// TwinCAT 3 PLC project PLC1
// ProgramVersion: 3.1.4026.16
// libraries:
//   Tc2_MC2, * (Beckhoff Automation GmbH)
//   Tc2_Standard, * (Beckhoff Automation GmbH)
//   Tc2_System, * (Beckhoff Automation GmbH)
// project tree:
//   DUTs/ E_State.TcDUT
//   / PlcTask.TcTTO
//   POUs/ eStopPLC.TcPOU, LightBar.TcPOU, MAIN.TcPOU, RevSeq.TcPOU
// real-time tasks:
//   TASK PlcTask: cycle T#10ms, priority 20, ADS port 350
// motion (NC):
//   TASK NC-Task 1 SAF: cycle T#2ms, priority 4, ADS port 501
//   TASK NC-Task 1 SVB: cycle T#10ms, priority 8, ADS port 511
//   AXIS Axis 1 (id 1)
//     General: UnitName=°
//     Dynamic: Acceleration=15000, Deceleration=15000, Jerk=145784.961
//     Velo: RefSearch=323.96658, RefSync=323.96658, SlowManual=1619.8329, FastManual=9718.9974, Fast=32396.658, Maximum=32396.658
//     OtherSettings: AllowMotionCmdToSlave=true
//     encoder EncType=19
//       EncPara: ScaleFactorNumerator=360, ScaleFactorDenominator=1048576, MaxCount=#xffffffff
//     drive DrvType=16
//       DrvPara: MaxCount=#xffffffff, DriveControlDWord=#x00000100
//         Analog: VeloReferenz=35636.3238, VeloScale=32, TorqueSetpointScale=10, ScaleFactorActTorque=0.1
//         TimeComp: TaskDelayCycles=1
//     controller CtrType=1
//       CtrPara: PriorControlFactor=1
//         Observer: BandWidth=20
// I/O:
//   DEVICE Device 1 (EtherCAT), AmsNetId 10.200.70.9.2.1
//     Term 1 (EK1200) [EK1200-5000 EtherCAT Power supply (2A E-Bus)]
//       Term 2 (EL1859) [EL1859 8Ch. Dig. Input 24V, 3ms, 8Ch. Dig. Output 24V, 0.5A]
//       Term 3 (EL1859) [EL1859 8Ch. Dig. Input 24V, 3ms, 8Ch. Dig. Output 24V, 0.5A]
//       Term 4 (EL3255) [EL3255 5Ch. potentiometer measurement with sensor supply]
//       Term 5 (EL3214-0090) [EL3214-0090 4Ch. Ana. Input PT100 (RTD), TwinSAFE SC]
//       Term 6 (EL5151) [EL5151 1Ch. Inc. Encoder]
//       Term 7 (EL1918) [EL1918, 8Ch. Safety Input 24V, TwinSAFE]
//         modules: Module 1 (FSOE), Module 2 (FSLOGIC)
//       Term 8 (EL2912) [EL2912, 2Ch. Safety Output 24V, 2A, TwinSAFE]
//         modules: Module 2 (FSOUT), Module 3 (DEVICEIO), Module 4 (FSLOGIC)
//       Term 9 (EL9110) [EL9110 Power Supplier with LED (24V, Diagnostics)]
//       Term 10 (EL7201-9014) [EL7201-9014 1Ch. MDP742 Servo motor output stage with OCT (50V, 2.8A RMS) and STO input]
//         startup 32784:18 := 0500
//         startup 32784:19 := B200
//         startup 32784:20 := 96000000
//         startup 32784:21 := 2B000000
//         startup 32785:17 := 98210000
//         startup 32785:18 := 960A0000
//         startup 32785:19 := 03
//         startup 32785:21 := 0E01
//         startup 32785:22 := 46000000
//         startup 32785:24 := 22000000
//         startup 32785:25 := 0F00
//         startup 32785:27 := F7120000
//         startup 32785:45 := 5501
//       Term 11 (EK1122) [EK1122 2 port EtherCAT junction]
//       Term 12 (EL9011) [EL9011 End Terminal]
// variable links:
//   (this object) <-> Device 1 (EtherCAT)/Term 1 (EK1200)/Term 10 (EL7201-9014)
//     Drive/Inputs/In/nDataIn1 <-> DRV Following error actual value/Following error actual value
//     Drive/Inputs/In/nDcOutputTime <-> InfoData/DcOutputShift
//     Drive/Inputs/In/nState1 <-> DRV Statusword/Statusword
//     Drive/Inputs/In/nState2 <-> DRV Statusword/Statusword @bit 8
//     Drive/Inputs/In/nState4 @bit 1 <-> WcState/InputToggle
//     Drive/Inputs/In/nState4 <-> WcState/WcState
//     Drive/Outputs/Out/nCtrl1 <-> DRV Controlword/Controlword
//     Drive/Outputs/Out/nCtrl2 <-> DRV Controlword/Controlword @bit 8
//     Drive/Outputs/Out/nDataOut1 <-> DRV Target position/Target position
//     Drive/Outputs/Out/nDataOut2 <-> DRV Target velocity/Target velocity
//     Enc/Inputs/In/nDataIn1 <-> FB Position/Position
//     Enc/Inputs/In/nDcInputTime <-> InfoData/DcInputShift
//     Enc/Inputs/In/nState4 @bit 1 <-> WcState/InputToggle
//     Enc/Inputs/In/nState4 <-> WcState/WcState
//   (this object) <-> Device 1 (EtherCAT)
//     Term 1 (EK1200)/Term 7 (EL1918)/Module 1 (FSOE)/FSoE Inputs/FSOE <-> Term 1 (EK1200)/Term 8 (EL2912)/ConnectionOutputs/Message_3 RxPDO
//     Term 1 (EK1200)/Term 7 (EL1918)/Module 1 (FSOE)/FSoE Outputs/FSOE <-> Term 1 (EK1200)/Term 8 (EL2912)/ConnectionInputs/Message_3 TxPDO
//     Term 1 (EK1200)/Term 8 (EL2912)/ConnectionInputs/Message_3 TxPDO <-> Term 1 (EK1200)/Term 7 (EL1918)/Module 1 (FSOE)/FSoE Outputs/FSOE
//     Term 1 (EK1200)/Term 8 (EL2912)/ConnectionOutputs/Message_3 RxPDO <-> Term 1 (EK1200)/Term 7 (EL1918)/Module 1 (FSOE)/FSoE Inputs/FSOE
//   PLC1 Instance <-> Device 1 (EtherCAT)/Term 1 (EK1200)/Term 2 (EL1859)
//     PlcTask Inputs/RevSeq.xEnable <-> Channel 4/Input
//     PlcTask Inputs/RevSeq.xReset <-> Channel 2/Input
//     PlcTask Inputs/RevSeq.xSetPos <-> Channel 3/Input
//     PlcTask Inputs/RevSeq.xStart <-> Channel 1/Input
//     PlcTask Inputs/eStopPLC.xSwitchSF14 <-> Channel 5/Input
//     PlcTask Inputs/eStopPLC.xSwitchSF15 <-> Channel 6/Input
//     PlcTask Outputs/LightBar.aLights[{1..8}] <-> Channel {9..16}/Output  (8 links)
//   PLC1 Instance <-> Device 1 (EtherCAT)/Term 1 (EK1200)/Term 4 (EL3255)
//     PlcTask Inputs/LightBar.iPot <-> AI Standard Channel 1/Value
//   PLC1 Instance <-> Device 1 (EtherCAT)/Term 1 (EK1200)/Term 8 (EL2912)
//     PlcTask Outputs/eStopPLC.xErrAck <-> StandardOutputs/Standard In Var 1
//     PlcTask Outputs/eStopPLC.xRun <-> StandardOutputs/Standard In Var 2
//   PLC1 Instance <-> NC-Task 1 SAF/Axes/Axis 1
//     PlcTask Inputs/RevSeq.Servo.NcToPlc <-> Outputs/ToPlc
//     PlcTask Outputs/RevSeq.Servo.PlcToNc <-> Inputs/FromPlc

CONFIGURATION PLC1
    RESOURCE PLC ON TwinCAT3
        TASK PlcTask(INTERVAL := T#10ms, PRIORITY := 20);
        PROGRAM MAIN WITH PlcTask : MAIN;
    END_RESOURCE
END_CONFIGURATION

// ---- DUTs/E_State.TcDUT
{attribute 'qualified_only'}
{attribute 'strict'}
{attribute 'to_string'}
TYPE E_State :
(
	Init,
	MovP1,
	WaitP1,
	MovP2,
	WaitP2,
	Error
);
END_TYPE

// ---- POUs/MAIN.TcPOU
PROGRAM MAIN
VAR
END_VAR

//Script written on 06/23/2025 for the CALA-TRCB stands in the LA office
//will need to activate config and download safeyt project

//test all lights on the stand
//turn potentiometer RA10 to turn all lights on and off
LightBar();

//motion test (drive manager 2 utalized
//switch 10 to power/enable the motor, switch 12 to reset errors, switch 13 to run through the motion
RevSeq();

//safety test (may need to delete previous safety projects to run)
//switch 14 to run and switch 15 to errAck
eStopPLC();

END_PROGRAM

// ---- POUs/LightBar.TcPOU
PROGRAM LightBar
VAR
	aLights AT %Q* : ARRAY [1..8] OF BOOL;
	
	iPot AT %I* : INT;
END_VAR

//turn all lights off
aLights[1] := aLights[2] := aLights[3] := aLights[4] := aLights[5] := aLights[6] := aLights[7] := aLights[8] := FALSE;

//turn lights on
CASE iPot OF
	0..10000:		//lights PF10 and PF11 on
		aLights[1] := aLights[2] := TRUE;
	10001..20000:	//lights PF10, PF11, PF12, PF13 on
		aLights[1] := aLights[2] := aLights[3] := aLights[4] := TRUE;
	20001..30000:	//lights PF10, PF11, PF12, PF13, PF14, PF15 on
		aLights[1] := aLights[2] := aLights[3] := aLights[4] := aLights[5] := aLights[6] := TRUE;
	30001..32767: 	//lights PF10, PF11, PF12, PF13, PF14, PF15, PF16, PF17 on
		aLights[1] := aLights[2] := aLights[3] := aLights[4] := aLights[5] := aLights[6] := aLights[7] := aLights[8] := TRUE;
END_CASE

END_PROGRAM

// ---- POUs/RevSeq.TcPOU
PROGRAM RevSeq
VAR
	//instance of the enumeration
	eState : E_State;
	
	//instances of MC2 FBs
	fbPower		: MC_Power;
	fbSetPos	: MC_SetPosition;
	fbMovAbs	: MC_MoveAbsolute;
	fbReset		: MC_Reset;
	
	Servo : AXIS_REF;
	
	//intalized variables
	lrOverRide  : LREAL := 100;
	lrSetPos	: LREAL := 0;
	
	//variable
	udiErrID : UDINT;
	
	lrP1 : LREAL;
	lrP2 : LREAL;
	lrV1 : LREAL;
	lrV2 : LREAL;
	
	tWait1 : TIME;
	tWait2 : TIME;
	
	//instance for a timer
	fbTimer : TON;
	
	xEnable AT %I* : BOOL;
	xStart AT %I* : BOOL;
	xReset AT %I*: BOOL;
	xSetPos AT %I*: BOOL;
	
END_VAR

//create PLCxEnableave reversing sequencexEnableoccur

//Outside of Case Statement
fbPower(
	Axis:= Servo, 
	Enable:= xEnable, 
	Enable_Positive:= xEnable, 
	Enable_Negative:= xEnable, 
	Override:= lrOverRide);
	
IF fbPower.Error THEN
	eState		:= E_State.Error;
	udiErrID	:= fbPower.ErrorID;
END_IF

//Case Statement
CASE eState OF
	E_State.Init:
		lrP1 := 1500;
		lrP2 := 9000;
		lrV1 := 7000;
		lrV2 := 4000;
		
		tWait1 := T#2S;
		tWait2 := T#5S;
		
		fbSetPos(
			Axis:= Servo, 
			Execute:= TRUE, 
			Position:= lrSetPos);
			
		IF fbPower.Status AND fbSetPos.Done AND xStart AND NOT xReset THEN
			eState := E_State.MovP1;
			fbSetPos(
				Axis:= Servo, 
				Execute:= FALSE); //function blocks need to be turned off to be able to use them again
		END_IF
		
		IF fbSetPos.Error THEN
			eState		:= E_State.Error;
			udiErrID	:= fbSetPos.ErrorID;
			fbSetPos(
				Axis:= Servo, 
				Execute:= FALSE);
		END_IF
	
	E_State.MovP1:
		fbMovAbs(
			Axis:= Servo, 
			Execute:= TRUE, 
			Position:= lrP1, 
			Velocity:= lrV1);
			
		IF fbMovAbs.Done THEN
			eState := E_State.WaitP1;
			fbMovAbs(
				Axis:= Servo, 
				Execute:= FALSE);
		END_IF
		
		IF fbMovAbs.Error THEN
			eState		:= E_State.Error;
			udiErrID	:= fbMovAbs.ErrorID;
			fbMovAbs(
				Axis:= Servo, 
				Execute:= FALSE);
		END_IF
	
	E_State.WaitP1:
		fbTimer(IN:= TRUE, PT:= tWait1);
			
		IF fbTimer.Q THEN
			eState := E_State.MovP2;
			fbTimer(IN:= FALSE);
		END_IF
	
	E_State.MovP2:
		fbMovAbs(
			Axis:= Servo, 
			Execute:= TRUE, 
			Position:= lrP2, 
			Velocity:= lrV2);
			
		IF fbMovAbs.Done THEN
			eState := E_State.WaitP2;
			fbMovAbs(
				Axis:= Servo, 
				Execute:= FALSE);
		END_IF
		
		IF fbMovAbs.Error THEN
			eState		:= E_State.Error;
			udiErrID	:= fbMovAbs.ErrorID;
			fbMovAbs(
				Axis:= Servo, 
				Execute:= FALSE);
		END_IF
	
	E_State.WaitP2:
		fbTimer(IN:= TRUE, PT:= tWait2);
			
		IF fbTimer.Q THEN
			eState := E_State.MovP1;
			fbTimer(IN:= FALSE);
		END_IF
	
	E_State.Error:
		fbReset(
			Axis:= Servo, 
			Execute:= xReset);
		
		IF fbReset.Done THEN
			eState := E_State.Init;
			fbSetPos(
				Axis:= Servo, 
				Execute:= FALSE);
			fbMovAbs(
				Axis:= Servo, 
				Execute:= FALSE);
			fbTimer(IN:= FALSE);
		END_IF

END_CASE

END_PROGRAM

// ---- POUs/eStopPLC.TcPOU
PROGRAM eStopPLC
VAR
	xSwitchSF14 AT %I* : BOOL;
	xSwitchSF15 AT %I* : BOOL;
	
	xRun 	AT %Q* : BOOL; 
	xErrAck AT %Q* : BOOL; 
END_VAR

xRun:= xSwitchSF14;
xErrAck := xSwitchSF15;

END_PROGRAM
